// TIA Portal V18 export
DATA_BLOCK "vessel"   // DB75
{ S7_Optimized_Access := 'TRUE' }
VERSION : 0.1
// stored: AutoNumber true, DBAccessibleFromOPCUA true, IsOnlyStoredInLoadMemory false, IsRetainMemResEnabled false, IsWriteProtectedInAS false, MemoryReserve 100
   VAR RETAIN
      "Duration pressure equalization" : Struct
         "A" : Int := 10;
         "B" : Int := 10;
      END_STRUCT;
      "amibient pressure" : Int := 900;
      "hysteresis ambient pressure" : Int := 50;
      "working pressure" : Struct
         "A" : Real := 3.0;
         "A+" : Real;
         "A-" : Real;
         "B" : Real := 3.0;
         "B+" : Real;
         "B-" : Real;
      END_STRUCT;
      "working pressure hysteresis" : Struct
         "A" : Real;
         "B" : Real;
      END_STRUCT;
   END_VAR
   VAR
      "Vaccum sensor selection" : Struct
         "selection A" : Int;
         "selection B" : Int;
         "A selected" : Bool;
         "B selected" : Bool;
         "A or B selected" : Bool;
      END_STRUCT;
      "Evacuation set Vaccum" : Struct
         A1 : Int;
         A2 : Int;
         B1 : Int;
         B2 : Int;
      END_STRUCT;
      "Evacuation Real vaccum" : Struct
         A1 : Int;
         A2 : Int;
         B1 : Int;
         B2 : Int;
      END_STRUCT;
      "Evacuation Time set" : Struct
         A1 : Int;
         A2 : Int;
         B1 : Int;
         B2 : Int;
      END_STRUCT;
      "Evacuation Time Real" : Struct
         A1 : Int;
         A2 : Int;
         B1 : Int;
         B2 : Int;
      END_STRUCT;
   END_VAR
   VAR RETAIN
      "preparation status" : Struct
         A1 : Int;
         A2 : Int;
         B1 : Int;
         B2 : Int;
      END_STRUCT;
      "monitor status" : Struct
         A1 : Int;
         A2 : Int;
         B1 : Int;
         B2 : Int;
      END_STRUCT;
      "Activate vessel" : Struct
         A1 : Bool;
         A2 : Bool;
         B1 : Bool;
         B2 : Bool;
      END_STRUCT;
   END_VAR
   VAR
      "A status" : Int;
      "B status" : Int;
   END_VAR
BEGIN
END_DATA_BLOCK
